FUNCTION_BLOCK A2X_LAST_2 (* MERGE 2 A2X in 1 A2X (LAST WRITER WINS je Kanal, nicht naiv gemergt) - UP und DOWN werden unabhaengig gemerged, welcher Socket zuletzt auf dem jeweiligen Kanal geschrieben hat, gewinnt *)
  (* Standard: 61499-2; Description: Copyright (c) 2026 Meisterschulen am Ostbahnhof This program and the accompanying materials are made available under the terms of the Eclipse Public License 2.0 which is available at https://www.eclipse.org/legal/epl-2.0/ SPDX-License-Identifier: EPL-2.0 *)
  (* Version 1.0, 2026-08-31, Franz Höpfinger, Meisterschulen am Ostbahnhof, 2-channel extension of the generic LAST_2 pattern - UP and DOWN are two independent single-channel merges sharing one ECC (only one event is processed per FB invocation, so no state collision) *)
  PACKAGE adapter::events::unidirectional;
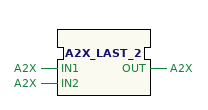
  SOCKETS
    IN1 : adapter::types::unidirectional::A2X;
    IN2 : adapter::types::unidirectional::A2X;
  END_SOCKETS
  PLUGS
    OUT : adapter::types::unidirectional::A2X;
  END_PLUGS
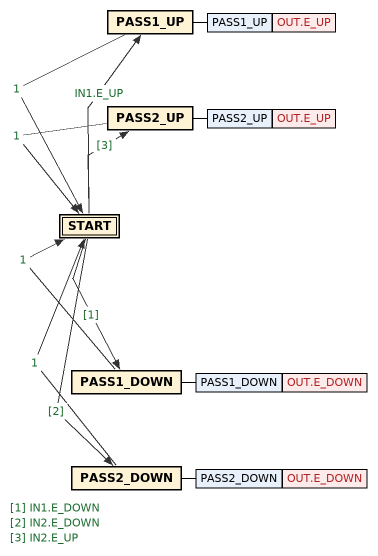
  EC_STATES
    START; (* Initial State *)
    PASS1_UP : PASS1_UP -> OUT.E_UP; (* IN1 zuletzt auf UP geschrieben *)
    PASS2_UP : PASS2_UP -> OUT.E_UP; (* IN2 zuletzt auf UP geschrieben *)
    PASS1_DOWN : PASS1_DOWN -> OUT.E_DOWN; (* IN1 zuletzt auf DOWN geschrieben *)
    PASS2_DOWN : PASS2_DOWN -> OUT.E_DOWN; (* IN2 zuletzt auf DOWN geschrieben *)
  END_STATES
  EC_TRANSITIONS
    START TO PASS1_UP := IN1.E_UP;
    START TO PASS2_UP := IN2.E_UP;
    START TO PASS1_DOWN := IN1.E_DOWN;
    START TO PASS2_DOWN := IN2.E_DOWN;
    PASS1_UP TO START := 1;
    PASS2_UP TO START := 1;
    PASS1_DOWN TO START := 1;
    PASS2_DOWN TO START := 1;
  END_TRANSITIONS
  ALGORITHM PASS1_UP IN ST: (* IN1.UP durchreichen *)
OUT.UP := IN1.UP;
  END_ALGORITHM
  ALGORITHM PASS2_UP IN ST: (* IN2.UP durchreichen *)
OUT.UP := IN2.UP;
  END_ALGORITHM
  ALGORITHM PASS1_DOWN IN ST: (* IN1.DOWN durchreichen *)
OUT.DOWN := IN1.DOWN;
  END_ALGORITHM
  ALGORITHM PASS2_DOWN IN ST: (* IN2.DOWN durchreichen *)
OUT.DOWN := IN2.DOWN;
  END_ALGORITHM
END_FUNCTION_BLOCK
